TYPE ST_EL7062 :
STRUCT
	//EtherCAT Terminal, 2-channel motion interface, stepper motor, 48 V DC
	Linear	:	ST_EL7062A1; //Axis 1 - Linear Pump 1 Amp (4600 steps limit)
	Rotary	:	ST_EL7062A2; //Axis 2 - Rotary pump 2 Amp (relative motion)
END_STRUCT
END_TYPE

(* stored: Version 1.1.0.1, ProductVersion 3.1.4024.12
   DUT ST_EL7062: Id {2e27b35d-596f-48e0-b292-3958049ff7df} *)
